Staubli VAL3: stopRobot.pgx

program stopRobot()
begin
  // mutex the motion status
  setMutex(cycleStatus:bMotionToken)
  cycleStatus:bWait=true
  stopMove()
  // check that the robot has been stopped
  if watch(cycleStatus:bMoveStopped==true,10)==false
    popUpMsg("error stopping the robot using an INPUT ")
    logMsg("error stopping the robot using an INPUT ")
    wait(cycleStatus:bMoveStopped==true)
  endIf
end
